// TIA Portal V19 export
TYPE "UDT_FMTOTALIZER"
   STRUCT
      trigger_add : Bool := false;
      trigger_force : Bool := false;
      trigger_reset : Bool := false;
      help_add : Bool := false;
      help_force : Bool := false;
      help_reset : Bool := false;
      cmd_add : Bool := false;
      cmd_force : Bool := false;
      cmd_reset : Bool := false;
      q_add_int : DInt := 0;
      q_add_dec : DInt := 0;
      q_total_int : DInt := 0;
      q_total_dec : DInt := 0;
      q_force_int : DInt := 0;
      q_force_dec : DInt := 0;
      q_max_dec : DInt := 0;
      q_total_real : Real := 0.0;
   END_STRUCT;
END_TYPE
